FUNCTION func_fac: DINT
VAR_INPUT
    farg_fac_a: DINT;
END_VAR

func_fac := ifExprFunc1(farg_fac_a);
RETURN;

END_FUNCTION

(* stored: ProductVersion 3.1.0.18, Version 1.1.0.1 *)
